# EPICS autosave request: iocBoot/obsolete/ioc13ida/auto_positions.req
file "CARS_8_motor_positions_sub.req",   P=$(P), M1=m33, M2=m34, M3=m35, M4=m36, M5=m37, M6=m38, M7=m39, M8=m40
file "CARS_8_motor_positions_sub.req",   P=$(P), M1=m41, M2=m42, M3=m43, M4=m44, M5=m45, M6=m46, M7=m47, M8=m48
file "CARS_8_motor_positions_sub.req",   P=$(P), M1=m49, M2=m50, M3=m51, M4=m52, M5=m53, M6=m54, M7=m55, M8=m56
